{attribute 'GeneratedUsingTerminal: EK1100-0000-0018'}
{attribute addProperty BoxType "EK1100-0000-0018"}
{attribute addProperty Id "Beckhoff_EL6xxxEK1122Beckhoff_EL6xxxEK1122_B6505ABE2A_0001_EL6001_0000_0000EL6001_DB28565A52A_0002_EL6001_0000_0016EL6001_0471BDA261A_0003_EL6001_0000_0017EL6001_0471BDA261A_0004_EL6001_0000_0018EL6001_0471BDA261A_0005_EL6001_0000_0019EL6001_0471BDA261A_0006_EL6001_0000_0020EL6001_0471BDA261A_0007_EL6002_0000_0016EL6002_44251D5B118A_0008_EL6002_0000_0017EL6002_C418D5E9118A_0009_EL6002_0000_0018EL6002_C418D5E9118A_0010_EL6002_0000_0019EL6002_C418D5E9118A_0011_EL6021_0000_0000EL6021_DB28565A52A_0012_EL6021_0000_0016EL6021_0471BDA261A_0013_EL6021_0000_0017EL6021_0471BDA261A_0014_EL6021_0000_0018EL6021_FC2726C561A_0015_EL6021_0000_0019EL6021_FC2726C561A_0016_EL6021_0000_0020EL6021_FC2726C561A_0017_EL6021_0000_0021EL6021_FC2726C561A_0018_EL6021_0021_0018EL6021_FC2726C561A_0019_EL6021_0021_0019EL6021_FC2726C561A_0020_EL6021_0021_0020EL6021_FC2726C561A_0021_EL6021_0021_0021EL6021_FC2726C561A_0022_EL6022_0000_0016EL6022_44251D5B118A_0023_EL6022_0000_0017EL6022_44251D5B118A_0024_EL6022_0000_0018EL6022_44251D5B118A_0025_EL6022_0000_0019EL6022_44251D5B118A_0026_EL6070_0000_0016EL6070_77C76A862A_0027_EL6070_0000_0017EL6070_77C76A862A_0028_EL6070_0000_0018EL6070_77C76A862A_0029_EL6070_0000_0019EL6070_77C76A862A_0030_EL6070_0033_0016EL6070_77C76A862A_0031_EL6070_0033_0017EL6070_77C76A862A_0032_EL6070_0033_0018EL6070_77C76A862A_0033_EL6070_0033_0019EL6070_77C76A862A_0034_EL6080_0000_0016EL6080_986F14164A_0035_EL6080_0000_0017EL6080_986F14164A_0036_EL6080_0000_0018EL6080_916B96A98A_0037_EL6080_0000_0020EL6080_916B96A98A_0038_EL6090_0000_0016EL6090_9BC1C0C414A_0039_EL6090_0000_0017EL6090_9BC1C0C414A_0040_EL6201_0000_0017EL6201_647A76CA516A_0041_EL6201_0000_0018EL6201_896BFBB2520A_0042_EL6201_0000_0019EL6201_896BFBB2520A_0043_EL6224_0000_0016EL6224_34BBFD238A_0044_EL6224_0000_0017EL6224_0B6584DB10A_0045_EL6224_0000_0018EL6224_0B6584DB10A_0046_EL6224_0000_0019EL6224_0B6584DB10A_0047_EL6224_0000_0020EL6224_0B6584DB10A_0048_EL6224_0000_0021EL6224_0B6584DB10A_0049_EL6224_0090_0016EL6224_21A73D0010A_0050_EL6224_0090_0017EL6224_21A73D0010"}
{attribute addProperty CRC "2226308695"}
{attribute addProperty Size "3667"}
TYPE Beckhoff_EL6xxx_84B2C657 EXTENDS EK1100_1FC0878B :
STRUCT
	{attribute addProperty Name "Beckhoff_EL6xxxEK1122"}
	{attribute addProperty PreviousPort "Beckhoff EL6xxx : B"}
	Beckhoff_EL6xxxEK1122 : Beckhoff_EL6xxxEK1122_B6505ABE;
	{attribute addProperty Name "A_0001_EL6001_0000_0000"}
	{attribute addProperty PreviousPort "Beckhoff EL6xxxEK1122 : C"}
	A_0001_EL6001_0000_0000 : EL6001_DB28565A;
	{attribute addProperty Name "A_0002_EL6001_0000_0016"}
	{attribute addProperty PreviousPort "A_0001(EL6001-0000-0000) : B"}
	A_0002_EL6001_0000_0016 : EL6001_0471BDA2;
	{attribute addProperty Name "A_0003_EL6001_0000_0017"}
	{attribute addProperty PreviousPort "A_0002(EL6001-0000-0016) : B"}
	A_0003_EL6001_0000_0017 : EL6001_0471BDA2;
	{attribute addProperty Name "A_0004_EL6001_0000_0018"}
	{attribute addProperty PreviousPort "A_0003(EL6001-0000-0017) : B"}
	A_0004_EL6001_0000_0018 : EL6001_0471BDA2;
	{attribute addProperty Name "A_0005_EL6001_0000_0019"}
	{attribute addProperty PreviousPort "A_0004(EL6001-0000-0018) : B"}
	A_0005_EL6001_0000_0019 : EL6001_0471BDA2;
	{attribute addProperty Name "A_0006_EL6001_0000_0020"}
	{attribute addProperty PreviousPort "A_0005(EL6001-0000-0019) : B"}
	A_0006_EL6001_0000_0020 : EL6001_0471BDA2;
	{attribute addProperty Name "A_0007_EL6002_0000_0016"}
	{attribute addProperty PreviousPort "A_0006(EL6001-0000-0020) : B"}
	A_0007_EL6002_0000_0016 : EL6002_44251D5B;
	{attribute addProperty Name "A_0008_EL6002_0000_0017"}
	{attribute addProperty PreviousPort "A_0007(EL6002-0000-0016) : B"}
	A_0008_EL6002_0000_0017 : EL6002_C418D5E9;
	{attribute addProperty Name "A_0009_EL6002_0000_0018"}
	{attribute addProperty PreviousPort "A_0008(EL6002-0000-0017) : B"}
	A_0009_EL6002_0000_0018 : EL6002_C418D5E9;
	{attribute addProperty Name "A_0010_EL6002_0000_0019"}
	{attribute addProperty PreviousPort "A_0009(EL6002-0000-0018) : B"}
	A_0010_EL6002_0000_0019 : EL6002_C418D5E9;
	{attribute addProperty Name "A_0011_EL6021_0000_0000"}
	{attribute addProperty PreviousPort "A_0010(EL6002-0000-0019) : B"}
	A_0011_EL6021_0000_0000 : EL6021_DB28565A;
	{attribute addProperty Name "A_0012_EL6021_0000_0016"}
	{attribute addProperty PreviousPort "A_0011(EL6021-0000-0000) : B"}
	A_0012_EL6021_0000_0016 : EL6021_0471BDA2;
	{attribute addProperty Name "A_0013_EL6021_0000_0017"}
	{attribute addProperty PreviousPort "A_0012(EL6021-0000-0016) : B"}
	A_0013_EL6021_0000_0017 : EL6021_0471BDA2;
	{attribute addProperty Name "A_0014_EL6021_0000_0018"}
	{attribute addProperty PreviousPort "A_0013(EL6021-0000-0017) : B"}
	A_0014_EL6021_0000_0018 : EL6021_FC2726C5;
	{attribute addProperty Name "A_0015_EL6021_0000_0019"}
	{attribute addProperty PreviousPort "A_0014(EL6021-0000-0018) : B"}
	A_0015_EL6021_0000_0019 : EL6021_FC2726C5;
	{attribute addProperty Name "A_0016_EL6021_0000_0020"}
	{attribute addProperty PreviousPort "A_0015(EL6021-0000-0019) : B"}
	A_0016_EL6021_0000_0020 : EL6021_FC2726C5;
	{attribute addProperty Name "A_0017_EL6021_0000_0021"}
	{attribute addProperty PreviousPort "A_0016(EL6021-0000-0020) : B"}
	A_0017_EL6021_0000_0021 : EL6021_FC2726C5;
	{attribute addProperty Name "A_0018_EL6021_0021_0018"}
	{attribute addProperty PreviousPort "A_0017(EL6021-0000-0021) : B"}
	A_0018_EL6021_0021_0018 : EL6021_FC2726C5;
	{attribute addProperty Name "A_0019_EL6021_0021_0019"}
	{attribute addProperty PreviousPort "A_0018(EL6021-0021-0018) : B"}
	A_0019_EL6021_0021_0019 : EL6021_FC2726C5;
	{attribute addProperty Name "A_0020_EL6021_0021_0020"}
	{attribute addProperty PreviousPort "A_0019(EL6021-0021-0019) : B"}
	A_0020_EL6021_0021_0020 : EL6021_FC2726C5;
	{attribute addProperty Name "A_0021_EL6021_0021_0021"}
	{attribute addProperty PreviousPort "A_0020(EL6021-0021-0020) : B"}
	A_0021_EL6021_0021_0021 : EL6021_FC2726C5;
	{attribute addProperty Name "A_0022_EL6022_0000_0016"}
	{attribute addProperty PreviousPort "A_0021(EL6021-0021-0021) : B"}
	A_0022_EL6022_0000_0016 : EL6022_44251D5B;
	{attribute addProperty Name "A_0023_EL6022_0000_0017"}
	{attribute addProperty PreviousPort "A_0022(EL6022-0000-0016) : B"}
	A_0023_EL6022_0000_0017 : EL6022_44251D5B;
	{attribute addProperty Name "A_0024_EL6022_0000_0018"}
	{attribute addProperty PreviousPort "A_0023(EL6022-0000-0017) : B"}
	A_0024_EL6022_0000_0018 : EL6022_44251D5B;
	{attribute addProperty Name "A_0025_EL6022_0000_0019"}
	{attribute addProperty PreviousPort "A_0024(EL6022-0000-0018) : B"}
	A_0025_EL6022_0000_0019 : EL6022_44251D5B;
	{attribute addProperty Name "A_0026_EL6070_0000_0016"}
	{attribute addProperty PreviousPort "A_0025(EL6022-0000-0019) : B"}
	A_0026_EL6070_0000_0016 : EL6070_77C76A86;
	{attribute addProperty Name "A_0027_EL6070_0000_0017"}
	{attribute addProperty PreviousPort "A_0026(EL6070-0000-0016) : B"}
	A_0027_EL6070_0000_0017 : EL6070_77C76A86;
	{attribute addProperty Name "A_0028_EL6070_0000_0018"}
	{attribute addProperty PreviousPort "A_0027(EL6070-0000-0017) : B"}
	A_0028_EL6070_0000_0018 : EL6070_77C76A86;
	{attribute addProperty Name "A_0029_EL6070_0000_0019"}
	{attribute addProperty PreviousPort "A_0028(EL6070-0000-0018) : B"}
	A_0029_EL6070_0000_0019 : EL6070_77C76A86;
	{attribute addProperty Name "A_0030_EL6070_0033_0016"}
	{attribute addProperty PreviousPort "A_0029(EL6070-0000-0019) : B"}
	A_0030_EL6070_0033_0016 : EL6070_77C76A86;
	{attribute addProperty Name "A_0031_EL6070_0033_0017"}
	{attribute addProperty PreviousPort "A_0030(EL6070-0033-0016) : B"}
	A_0031_EL6070_0033_0017 : EL6070_77C76A86;
	{attribute addProperty Name "A_0032_EL6070_0033_0018"}
	{attribute addProperty PreviousPort "A_0031(EL6070-0033-0017) : B"}
	A_0032_EL6070_0033_0018 : EL6070_77C76A86;
	{attribute addProperty Name "A_0033_EL6070_0033_0019"}
	{attribute addProperty PreviousPort "A_0032(EL6070-0033-0018) : B"}
	A_0033_EL6070_0033_0019 : EL6070_77C76A86;
	{attribute addProperty Name "A_0034_EL6080_0000_0016"}
	{attribute addProperty PreviousPort "A_0033(EL6070-0033-0019) : B"}
	A_0034_EL6080_0000_0016 : EL6080_986F1416;
	{attribute addProperty Name "A_0035_EL6080_0000_0017"}
	{attribute addProperty PreviousPort "A_0034(EL6080-0000-0016) : B"}
	A_0035_EL6080_0000_0017 : EL6080_986F1416;
	{attribute addProperty Name "A_0036_EL6080_0000_0018"}
	{attribute addProperty PreviousPort "A_0035(EL6080-0000-0017) : B"}
	A_0036_EL6080_0000_0018 : EL6080_916B96A9;
	{attribute addProperty Name "A_0037_EL6080_0000_0020"}
	{attribute addProperty PreviousPort "A_0036(EL6080-0000-0018) : B"}
	A_0037_EL6080_0000_0020 : EL6080_916B96A9;
	{attribute addProperty Name "A_0038_EL6090_0000_0016"}
	{attribute addProperty PreviousPort "A_0037(EL6080-0000-0020) : B"}
	A_0038_EL6090_0000_0016 : EL6090_9BC1C0C4;
	{attribute addProperty Name "A_0039_EL6090_0000_0017"}
	{attribute addProperty PreviousPort "A_0038(EL6090-0000-0016) : B"}
	A_0039_EL6090_0000_0017 : EL6090_9BC1C0C4;
	{attribute addProperty Name "A_0040_EL6201_0000_0017"}
	{attribute addProperty PreviousPort "A_0039(EL6090-0000-0017) : B"}
	A_0040_EL6201_0000_0017 : EL6201_647A76CA;
	{attribute addProperty Name "A_0041_EL6201_0000_0018"}
	{attribute addProperty PreviousPort "A_0040(EL6201-0000-0017) : B"}
	A_0041_EL6201_0000_0018 : EL6201_896BFBB2;
	{attribute addProperty Name "A_0042_EL6201_0000_0019"}
	{attribute addProperty PreviousPort "A_0041(EL6201-0000-0018) : B"}
	A_0042_EL6201_0000_0019 : EL6201_896BFBB2;
	{attribute addProperty Name "A_0043_EL6224_0000_0016"}
	{attribute addProperty PreviousPort "A_0042(EL6201-0000-0019) : B"}
	A_0043_EL6224_0000_0016 : EL6224_34BBFD23;
	{attribute addProperty Name "A_0044_EL6224_0000_0017"}
	{attribute addProperty PreviousPort "A_0043(EL6224-0000-0016) : B"}
	A_0044_EL6224_0000_0017 : EL6224_0B6584DB;
	{attribute addProperty Name "A_0045_EL6224_0000_0018"}
	{attribute addProperty PreviousPort "A_0044(EL6224-0000-0017) : B"}
	A_0045_EL6224_0000_0018 : EL6224_0B6584DB;
	{attribute addProperty Name "A_0046_EL6224_0000_0019"}
	{attribute addProperty PreviousPort "A_0045(EL6224-0000-0018) : B"}
	A_0046_EL6224_0000_0019 : EL6224_0B6584DB;
	{attribute addProperty Name "A_0047_EL6224_0000_0020"}
	{attribute addProperty PreviousPort "A_0046(EL6224-0000-0019) : B"}
	A_0047_EL6224_0000_0020 : EL6224_0B6584DB;
	{attribute addProperty Name "A_0048_EL6224_0000_0021"}
	{attribute addProperty PreviousPort "A_0047(EL6224-0000-0020) : B"}
	A_0048_EL6224_0000_0021 : EL6224_0B6584DB;
	{attribute addProperty Name "A_0049_EL6224_0090_0016"}
	{attribute addProperty PreviousPort "A_0048(EL6224-0000-0021) : B"}
	A_0049_EL6224_0090_0016 : EL6224_21A73D00;
	{attribute addProperty Name "A_0050_EL6224_0090_0017"}
	{attribute addProperty PreviousPort "A_0049(EL6224-0090-0016) : B"}
	A_0050_EL6224_0090_0017 : EL6224_21A73D00;
END_STRUCT
END_TYPE

(* stored: Version 1.2.0.0, ProductVersion 3.1.4024.9
   DUT Beckhoff_EL6xxx_84B2C657: Id {2f0dff61-6b6c-4217-820e-268549e91484} *)
